FUNCTION_BLOCK URMSGmonitoring (* Tamplate for a simple Basic Function Block Type *)
  (* Standard: 61499-2 *)
  (* Version 0.0, 2018-03-05, 4DIAC-IDE, 4DIAC-Consortium *)
  (* Version 1.0, 2016-05-26, AZ, fortiss GmbH *)
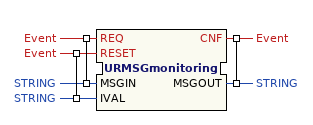
  EVENT_INPUT
    REQ WITH MSGIN; (* Normal Execution Request *)
    RESET WITH IVAL;
  END_EVENT
  EVENT_OUTPUT
    CNF WITH MSGOUT; (* Execution Confirmation *)
  END_EVENT
  VAR_INPUT
    MSGIN : STRING; (* Input event qualifier *)
    IVAL : STRING;
  END_VAR
  VAR_OUTPUT
    MSGOUT : STRING; (* Output event qualifier *)
  END_VAR
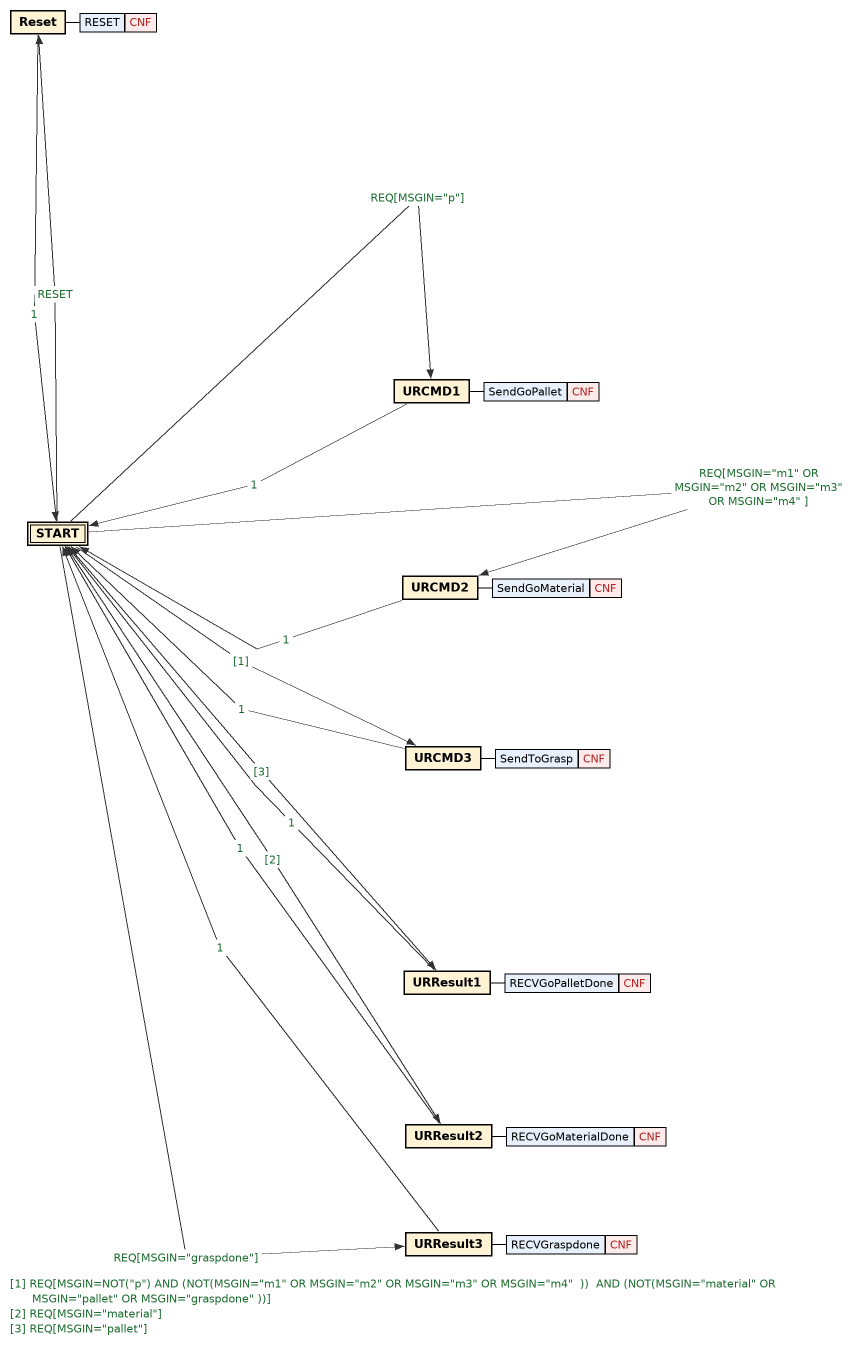
  EC_STATES
    START; (* Initial State *)
    URCMD1 : SendGoPallet -> CNF;
    URCMD2 : SendGoMaterial -> CNF;
    URCMD3 : SendToGrasp -> CNF;
    URResult1 : RECVGoPalletDone -> CNF;
    URResult2 : RECVGoMaterialDone -> CNF;
    URResult3 : RECVGraspdone -> CNF;
    Reset : RESET -> CNF;
  END_STATES
  EC_TRANSITIONS
    START TO URCMD3 := REQ[MSGIN=NOT("p") AND (NOT(MSGIN="m1" OR MSGIN="m2" OR MSGIN="m3" OR MSGIN="m4"  ))  AND (NOT(MSGIN="material" OR MSGIN="pallet" OR MSGIN="graspdone" ))];
    START TO URCMD2 := REQ[MSGIN="m1" OR MSGIN="m2" OR MSGIN="m3" OR MSGIN="m4" ];
    START TO URCMD1 := REQ[MSGIN="p"];
    URCMD3 TO START := 1;
    URCMD2 TO START := 1;
    URCMD1 TO START := 1;
    START TO URResult1 := REQ[MSGIN="pallet"];
    URResult1 TO START := 1;
    START TO URResult2 := REQ[MSGIN="material"];
    URResult2 TO START := 1;
    START TO URResult3 := REQ[MSGIN="graspdone"];
    URResult3 TO START := 1;
    START TO Reset := RESET;
    Reset TO START := 1;
  END_TRANSITIONS
  ALGORITHM SendGoPallet IN ST: (* new algorithm *)
MSGOUT:="GoPallet";
  END_ALGORITHM
  ALGORITHM SendGoMaterial IN ST: (* new algorithm *)
MSGOUT:=MSGIN;
  END_ALGORITHM
  ALGORITHM SendToGrasp IN ST: (* new algorithm *)
MSGOUT:=MSGIN;
  END_ALGORITHM
  ALGORITHM RECVGoPalletDone IN ST: (* new algorithm *)
MSGOUT:="UR arrives at pallet!";
  END_ALGORITHM
  ALGORITHM RECVGoMaterialDone IN ST: (* new algorithm *)
MSGOUT:="UR arrives at material zone";
  END_ALGORITHM
  ALGORITHM RECVGraspdone IN ST: (* new algorithm *)
MSGOUT:="UR Grasp Done!";
  END_ALGORITHM
  ALGORITHM RESET IN ST: (* new algorithm *)
MSGOUT:=IVAL;
  END_ALGORITHM
END_FUNCTION_BLOCK
